// TIA Portal V20 export
TYPE "typeCmControlNodeInterlock"
// stored: Namespace Unit1.Em9
   STRUCT
      visionStageLift : "LER_typeTwoWayActuatorInterlock";
      visionLight : "LER_typeTwoWayActuatorInterlock";
   END_STRUCT;
END_TYPE
